# EPICS substitutions: vacuum/MAIN_TRUNK/db/su3_agilent4uhv.substitutions
# Agilent4UHV substitutions file

file db/agilent4uhv.db
{
     pattern {LOCA,			DEV,		PORT,		ADDR,	TIMEOUT}
     		 {SU1,			SU3,		4uhv_1,		0,		0.2}
}
file db/agilent4uhv_alias.db
{
     pattern {LOCA,			DEV,		SUB1,					SUB2,					SUB3,						SUB4,				PORT,	ADDR,	TIMEOUT}
     		 {SU1,			SU3,	VU401:IP01:SIP20,	VU402:IP01:SIP20,		 VSS:IP01:SIP20,			VU403:IP01:SIP20,	4uhv_1,	0,		0.2}
}
